PROGRAM MAIN
VAR
	// Define EPICS interface for moving motor (struct)
	{attribute 'pytmc' := 'pv: TST:PLC-MOTION'}
	{attribute 'TcLinkTo' := '.nRawEncoderULINT     := TIID^Device 1 (EtherCAT)^Term 1 (EK1200)^Term 4 (EL5042)^FB Inputs Channel 1^Position'}
	M1: ST_MotionStage := (sName := 'MOTION:PRACTICE',
                        bPowerSelf := True); // opt out of PMPS and handle
											// motor enabling within FB_MotionStage
	
	// Attribute Linking (for hardware)
	// Inputs (Limit Switch)
	{attribute 'TcLinkTo' := 'TIID^Device 1 (EtherCAT)^Term 1 (EK1200)^Term 3 (EL1084)^Channel 1^Input'}
	backwardLimitSwitch AT %I* : BOOL;
	
	{attribute 'TcLinkTo' := 'TIID^Device 1 (EtherCAT)^Term 1 (EK1200)^Term 3 (EL1084)^Channel 2^Input'}
	forwardLimitSwitch AT %I* : BOOL;
	
	// Function Block Logic 
	fbMotion1: FB_MotionStage;

END_VAR

// Limit switch is NPN, while motion library uses PNP
M1.bLimitForwardEnable := NOT forwardLimitSwitch;
M1.bLimitBackwardEnable := NOT backwardLimitSwitch;

M1.bHardwareEnable := TRUE; // ok to move

// Invoke function block call
fbMotion1(stMotionStage := M1);

END_PROGRAM

(* stored: Version 1.1.0.1, ProductVersion 3.1.4024.12
   POU MAIN: Id {622f6e59-0aa4-465f-9317-a2a4d783d5c1}, SpecialFunc None *)
